// TIA Portal V17 export
// export: Created 2022-07-28T18:02:50.6515825Z, ExportSetting None, DisplayName Totally Integrated Automation Portal, DisplayVersion V17, DisplayName TIA Portal Openness, DisplayVersion V17, DisplayName TIA Portal Teamcenter Gateway, DisplayVersion V17, DisplayName TIA Portal Version Control Interface, DisplayVersion V17, DisplayName TIA Portal Test Suite Advanced, DisplayVersion V17, DisplayName SINAMICS Startdrive Advanced, DisplayVersion V17, DisplayName SINAMICS DCC, DisplayVersion V17, DisplayName SINAMICS Startdrive G130, G150, S120, S150, SINAMICS MV, S210, DisplayVersion V17, DisplayName SINAMICS Startdrive G110M, G120, G120C, G120D, G120P, G115D, DisplayVersion V17, DisplayName STEP 7 Professional, DisplayVersion V17, DisplayName SIMATIC Energy Suite, DisplayVersion V17, DisplayName STEP 7 CFC, DisplayVersion V17, DisplayName STEP 7 Safety, DisplayVersion V17, DisplayName WinCC Advanced / Unified PC, DisplayVersion V17, DisplayName SIMATIC Visualization Architect, DisplayVersion V17
FUNCTION_BLOCK "lib_fb_DSensor"   // FB18, SCL
{ S7_Optimized_Access := 'TRUE' }
AUTHOR : bean
// Descrete sensor functional block
// stored: MemoryReserve 100, SetENOAutomatically false
   VAR_INPUT
      I_Initialization { ExternalAccessible := 'False'; ExternalVisible := 'False'; ExternalWritable := 'False'} : Bool := FALSE;   // 1 = Restart PLC is active (First scan)
      I_Raw { ExternalAccessible := 'False'; ExternalVisible := 'False'; ExternalWritable := 'False'} : Bool;   // Sensor input
      II_Mode { ExternalAccessible := 'False'; ExternalVisible := 'False'; ExternalWritable := 'False'} : Int := -1;   // Check input: 0 - NO fault, 1 - NC fault, 2 - NO warning, 3 - NC warning, 4 - NO Info condition? 5 - NC Info condition
      I_GlobalRST { ExternalAccessible := 'False'; ExternalVisible := 'False'; ExternalWritable := 'False'} : Bool;   // Reset faults
      IR_CycleTime { ExternalAccessible := 'False'; ExternalVisible := 'False'; ExternalWritable := 'False'} : Real;   // PLC last cycle time
      II_Obj_ID { ExternalAccessible := 'False'; ExternalVisible := 'False'; ExternalWritable := 'False'} : Int := -1;   // Tech ID of object
   END_VAR
   VAR_OUTPUT
      Q_ProccessedVal { ExternalAccessible := 'False'; ExternalVisible := 'False'; ExternalWritable := 'False'} : Bool;   // Proccessed value by time and modes
      Q_FLT { ExternalAccessible := 'False'; ExternalVisible := 'False'; ExternalWritable := 'False'} : Bool;   // Fault is active
      Q_WRN { ExternalAccessible := 'False'; ExternalVisible := 'False'; ExternalWritable := 'False'} : Bool;   // Warning is active
      Q_INFO { ExternalAccessible := 'False'; ExternalVisible := 'False'; ExternalWritable := 'False'} : Bool;   // Info condition is active
      Q_DBReadErr { ExternalAccessible := 'False'; ExternalVisible := 'False'; ExternalWritable := 'False'} : Bool;   // Object DB reading fault
   END_VAR
   VAR_IN_OUT
      IO_PLC_CycleInfo : Variant;
   END_VAR
   VAR
      s_SimMode { ExternalAccessible := 'False'; ExternalVisible := 'False'; ExternalWritable := 'False'} : Bool;   // Simulation mode is active
      s_Suppressed { ExternalAccessible := 'False'; ExternalVisible := 'False'; ExternalWritable := 'False'} : Bool;   // Suppress fault/warning
      TON_FLT { ExternalAccessible := 'False'; ExternalVisible := 'False'; ExternalWritable := 'False'} : "Lib_FB_Timer_ON_Simple";
      EdgeError { ExternalAccessible := 'False'; ExternalVisible := 'False'; ExternalWritable := 'False'} : "Lib_FB_Edge";
      EdgeWarning { ExternalAccessible := 'False'; ExternalVisible := 'False'; ExternalWritable := 'False'} : "Lib_FB_Edge";
   END_VAR
   VAR RETAIN
      s_Obj_Retain_BUp { ExternalAccessible := 'False'; ExternalVisible := 'False'; ExternalWritable := 'False'} : Struct
         Config : "_DSensor_Config";
         s_Suppressed : Bool;   // Suppress faults
      END_STRUCT;
      s_Simulation { ExternalAccessible := 'False'; ExternalVisible := 'False'; ExternalWritable := 'False'} : Struct
         Obj_DATA_BACKUP : Struct
            Config : "_DSensor_Config";
            s_Suppressed { S7_SetPoint := 'True'} : Bool;   // Suppress faults
         END_STRUCT;
      END_STRUCT;
   END_VAR
   VAR_TEMP
      t_FltMode : Bool;   // 1 - Fault mode is active
      t_WarnMode : Bool;   // 1 - Warn mode is active
      t_InfoMode : Bool;   // 1 - Info mode is active
      t_RST_FLT : Bool;
      t_DBReadErr : Bool;   // Fault while DB reading
      ti_DBReadErr : Int;   // Fault # while DB reading
      ti_CMDLogic : Int;   // Command word for logic
      ti_NumObjDB : UInt;   // Number of DB for storage object data
      t_ObjAnyHMI : DB_ANY;   // Ref to object data
      t_ObjVarHMI : Variant;   // Ref to object data
      t_ObjAnyPLC : DB_ANY;   // Ref to object data
      t_ObjVarPLC : Variant;   // Ref to object data
      tud_DB_ShiftHMI : UInt;   // HMI object DB number shift
      tud_DB_ShiftPLC : UInt;   // PLC object DB number shift
      t_PLC_CycleInfo : "Lib_PLC_CycleInfo";
      t_Obj_HMI : "lib_udt_DSensor_HMI";
      t_Obj_PLC : "lib_udt_DSensor_PLC";
   END_VAR
BEGIN
   //Check input:
   //0 - NO fault,
   //1 - NC fault,
   //2 - NO warning,
   //3 - NC warning,
   //4 - NO Info condition,
   //5 - NC Info condition
   //
   REGION Inputs  
       //Reinit tempory variables
       REGION Reinit tempory variables


       END_REGION

       VariantGet(SRC := #IO_PLC_CycleInfo,
                  DST => #t_PLC_CycleInfo);

       //Read Object data
       //Reinit temp values
       #t_Obj_HMI := "D_ZeroTypes".DSensor_HMI;
       #t_Obj_PLC := "D_ZeroTypes".DSensor_PLC;
       #tud_DB_ShiftHMI := "D_General_ProgramDATA".ui_Shift_DBSens_HMI;
       #tud_DB_ShiftPLC := "D_General_ProgramDATA".ui_Shift_DBSens_PLC;
       #t_FltMode := false;
       #t_WarnMode := false;
       #t_InfoMode := false;

       IF #II_Obj_ID >= 0
       THEN
           #ti_NumObjDB := INT_TO_UINT(#II_Obj_ID) + #tud_DB_ShiftHMI;
           #t_ObjAnyHMI := UINT_TO_DB_ANY(#ti_NumObjDB);
           #t_ObjVarHMI := DB_ANY_TO_VARIANT(in := #t_ObjAnyHMI, err => #ti_DBReadErr);

           //If DB exist and convertion without error
           IF #ti_DBReadErr = 0
           THEN
               VariantGet(SRC := #t_ObjVarHMI,
                          DST => #t_Obj_HMI);
           ELSE
               #t_DBReadErr := true;
           END_IF;

           #ti_NumObjDB := INT_TO_UINT(#II_Obj_ID)+ #tud_DB_ShiftPLC;
           #t_ObjAnyPLC := UINT_TO_DB_ANY(#ti_NumObjDB);
           #t_ObjVarPLC := DB_ANY_TO_VARIANT(in := #t_ObjAnyPLC, err => #ti_DBReadErr);

           //If DB exist and convertion without error
           IF #ti_DBReadErr = 0
           THEN
               VariantGet(SRC := #t_ObjVarPLC,
                          DST => #t_Obj_PLC);
           ELSE
               #t_DBReadErr := true;
           END_IF;

       ELSE
           #t_DBReadErr := true;
       END_IF;


       //Read retain data if initialization is active
       IF #I_Initialization
       THEN
           #t_Obj_HMI.Config := #s_Obj_Retain_BUp.Config;
           #s_Suppressed := #s_Obj_Retain_BUp.s_Suppressed;
       END_IF;

       //Define CMD by priority
       IF #t_PLC_CycleInfo.CMD_GLOBAL <> 0
       THEN
           #ti_CMDLogic := #t_PLC_CycleInfo.CMD_GLOBAL;
       ELSE
           IF #t_Obj_HMI.CMD <> 0
           THEN
               #ti_CMDLogic := #t_Obj_HMI.CMD;
               #t_Obj_HMI.CMD := 0;
           END_IF;
       END_IF;

       #t_RST_FLT := #I_GlobalRST
       OR #t_Obj_HMI.Config.AutoReset;

       CASE #ti_CMDLogic OF
           0:  //Do nothing
               ;
           7:  //Sim mode ON
               IF NOT #s_SimMode
               THEN
                   #s_SimMode := TRUE;
                   #s_Simulation.Obj_DATA_BACKUP.Config := #t_Obj_HMI.Config;
                   #s_Simulation.Obj_DATA_BACKUP.s_Suppressed := #s_Suppressed;
               END_IF;
           8:  //Sim mode OFF
               IF #s_SimMode
               THEN
                   #s_SimMode := FALSE;
                   #t_Obj_HMI.Config := #s_Simulation.Obj_DATA_BACKUP.Config;
                   #s_Suppressed := #s_Simulation.Obj_DATA_BACKUP.s_Suppressed;
               END_IF;
           31..32://Reset faults
               #t_RST_FLT := TRUE;
           34: //Set bit for autoreset output 
               #t_Obj_HMI.Config.AutoReset := true;
           35: //Reset bit for autoreset output 
               #t_Obj_HMI.Config.AutoReset := false;
           64: //Fault/warning suppressed
               #s_Suppressed := NOT #s_Suppressed;
           80: //Discrete sensor. Invert value (Sim Mode)
               IF #s_SimMode
               THEN
                   #t_Obj_PLC.State.DisplayData := NOT #t_Obj_PLC.State.DisplayData;
               END_IF;
           ELSE//
               ;
       END_CASE;

   END_REGION

   REGION Proccess output value by mode
       #t_Obj_PLC.State.SensorValueHW := #I_Raw
       AND NOT #s_SimMode;

       CASE #II_Mode OF
           0:  //NO Fault condition
               #t_Obj_PLC.State.SensorValueLogic := #t_Obj_PLC.State.SensorValueHW;
               #t_FltMode := true;
               #t_Obj_PLC.State.SensorNO := true;
           1:  //NC Fault condition
               #t_Obj_PLC.State.SensorValueLogic := NOT #t_Obj_PLC.State.SensorValueHW;
               #t_FltMode := true;
               #t_Obj_PLC.State.SensorNO := false;
           2:  //NO Warning condition
               #t_Obj_PLC.State.SensorValueLogic := #t_Obj_PLC.State.SensorValueHW;
               #t_WarnMode := true;
               #t_Obj_PLC.State.SensorNO := true;
           3:  //NC Warning condition
               #t_Obj_PLC.State.SensorValueLogic := NOT #t_Obj_PLC.State.SensorValueHW;
               #t_WarnMode := true;
               #t_Obj_PLC.State.SensorNO := false;
           4:  //NO Info condition
               #t_Obj_PLC.State.SensorValueLogic := #t_Obj_PLC.State.SensorValueHW;
               #t_InfoMode := true;
               #t_Obj_PLC.State.SensorNO := true;
           5:  //NC Info condition
               #t_Obj_PLC.State.SensorValueLogic := NOT #t_Obj_PLC.State.SensorValueHW;
               #t_InfoMode := true;
               #t_Obj_PLC.State.SensorNO := false;
           ELSE  //
               #t_Obj_HMI := "D_ZeroTypes".DSensor_HMI;
               #t_Obj_PLC := "D_ZeroTypes".DSensor_PLC;

               IF NOT #t_DBReadErr THEN
                   VariantPut(SRC := #t_Obj_HMI,
                              DST := #t_ObjVarHMI);

                   VariantPut(SRC := #t_Obj_PLC,
                              DST := #t_ObjVarPLC);
               END_IF;

               #Q_ProccessedVal :=
               #Q_FLT :=
               #Q_WRN :=
               #Q_INFO := false;
               #Q_DBReadErr := true;

               RETURN;
       END_CASE;
       REGION Warnings and faults 
           //Time befor out detect
           #TON_FLT(IB_StartTimerInput := #t_Obj_PLC.State.SensorValueLogic,
                    IR_CycleTime := #IR_CycleTime,
                    IR_SpTime := #t_Obj_HMI.Config.WarnDetectTime);

           //Proccessed output value
           IF NOT #s_SimMode
           THEN
               #t_Obj_PLC.State.DisplayData := (#TON_FLT.QB_TimerOut
               OR (#t_Obj_PLC.State.DisplayData
               AND NOT #t_RST_FLT))
               AND NOT #s_Suppressed;
           ELSE
               #t_Obj_PLC.State.DisplayData := #t_Obj_PLC.State.DisplayData;
           END_IF;

           #t_Obj_PLC.State.SomeFlt := #t_Obj_PLC.State.DisplayData
           AND  #t_FltMode;

           #t_Obj_PLC.State.SomeWrn := #t_Obj_PLC.State.DisplayData
           AND #t_WarnMode;

           #t_Obj_PLC.State.SomeInfo := #t_Obj_PLC.State.DisplayData
           AND #t_InfoMode;

           //Excluded (suppressed) fault is active
           #t_Obj_PLC.State.SuppressedFltWrn := (#TON_FLT.QB_TimerOut
           AND #s_Suppressed);

           //New fault checking
           #EdgeError(IB_Input := #t_Obj_PLC.State.SomeFlt);
           //New warning checking
           #EdgeWarning(IB_Input := #t_Obj_PLC.State.SomeWrn);

       END_REGION
   END_REGION

   REGION PLC State + Counter
       "Lib_FC_DSens_CycleInfo_Count_State"(Alarm := #t_Obj_PLC.State.SomeFlt,
                                            AlarmNew := #EdgeError.QB_EdgePos,
                                            Warning := #t_Obj_PLC.State.SomeWrn,
                                            WarningNew := #EdgeWarning.QB_EdgePos,
                                            Simulation := #s_SimMode,
                                            PLC_CycleInfo := #t_PLC_CycleInfo);

   END_REGION

   REGION Write retain data to BUp
       //Read retain data if initialization is active
       IF NOT #I_Initialization
       THEN
           #s_Obj_Retain_BUp.Config :=  #t_Obj_HMI.Config;
           #s_Obj_Retain_BUp.s_Suppressed := #s_Suppressed;
       END_IF;
   END_REGION


   REGION Outputs
       //Outputs
       //Object DBs
       //HMI DB
       #t_Obj_HMI.CMD := 0;

       #t_Obj_HMI.ID := #II_Obj_ID;
       #t_Obj_HMI.CLSID := 40;

       //Write alarms to PLC storage
       #t_Obj_PLC.Alarm.SensorFlt := #t_Obj_PLC.State.SomeFlt;
       #t_Obj_PLC.Alarm.SensorWrn := #t_Obj_PLC.State.SomeWrn;
       #t_Obj_PLC.Alarm.SensorInfo := #t_Obj_PLC.State.SomeInfo;
       #t_Obj_PLC.Alarm.SimMode := #s_SimMode;
       #t_Obj_PLC.Alarm.NotSimMode := NOT #s_SimMode;
       #t_Obj_PLC.Alarm.Suppressed := #s_Suppressed;
       #t_Obj_PLC.Alarm.Consider := NOT #s_Suppressed;
       #t_Obj_PLC.Alarm.AutoResetEn := #t_Obj_PLC.State.AutoReset;
       #t_Obj_PLC.Alarm.AutoResetDis := NOT #t_Obj_PLC.State.AutoReset;
       #t_Obj_PLC.Alarm.SuppesedActive := #t_Obj_PLC.State.SuppressedFltWrn;

       //Write alarms to HMI
       #t_Obj_HMI.Status.w_AW1.%X0 := #t_Obj_PLC.Alarm.SensorFlt;       //х0 - Sensor Fault signal
       #t_Obj_HMI.Status.w_AW1.%X1 := #t_Obj_PLC.Alarm.SensorWrn;          //х1 - Sensor Warning signal
       #t_Obj_HMI.Status.w_AW1.%X2 := #t_Obj_PLC.Alarm.SensorInfo;         //x2 - Sensor Info signal
       #t_Obj_HMI.Status.w_AW1.%X3 := #t_Obj_PLC.Alarm.SimMode;      //x3 - Sim mode is active
       #t_Obj_HMI.Status.w_AW1.%X4 := NOT #t_Obj_PLC.Alarm.NotSimMode;  //x4 - Sim mode disabled
       #t_Obj_HMI.Status.w_AW1.%X5 := #t_Obj_PLC.Alarm.SuppesedActive; //x5 - Suppressed value is active

       #t_Obj_HMI.Status.w_AW2.%X0 := #t_Obj_PLC.Alarm.Suppressed;       //х0 - Suppress fault/warning
       #t_Obj_HMI.Status.w_AW2.%X1 := #t_Obj_PLC.Alarm.Consider;   //x1 - Consider fault/warning
       #t_Obj_HMI.Status.w_AW2.%X2 := #t_Obj_PLC.Alarm.AutoResetEn;       //х0 - Suppress fault/warning
       #t_Obj_HMI.Status.w_AW2.%X3 := #t_Obj_PLC.Alarm.AutoResetDis;   //x1 - Consider fault/warning

       //Write STW to PLC storage
       #t_Obj_PLC.State.AutoReset := #t_Obj_HMI.Config.AutoReset;
       #t_Obj_PLC.State.SimMode := #s_SimMode;
       #t_Obj_PLC.State.ReadFlt := #t_DBReadErr;
       #t_Obj_PLC.State.SuppressFltWrn := #s_Suppressed;

       //Write STW to HMI
       #t_Obj_HMI.Status.dw_STW.%X0  :=  #t_Obj_PLC.State.DisplayData;
       #t_Obj_HMI.Status.dw_STW.%X1  :=  #t_Obj_PLC.State.SimMode;
       #t_Obj_HMI.Status.dw_STW.%X2  :=  #t_Obj_PLC.State.SomeFlt;
       #t_Obj_HMI.Status.dw_STW.%X3  :=  #t_Obj_PLC.State.SomeWrn;
       #t_Obj_HMI.Status.dw_STW.%X4  :=  #t_Obj_PLC.State.SomeInfo;
       #t_Obj_HMI.Status.dw_STW.%X5  :=  #t_Obj_PLC.State.SuppressedFltWrn;
       #t_Obj_HMI.Status.dw_STW.%X6  :=  #t_Obj_PLC.State.ReadFlt;
       #t_Obj_HMI.Status.dw_STW.%X7  :=  #t_Obj_PLC.State.SuppressFltWrn;
       #t_Obj_HMI.Status.dw_STW.%X8  :=  #t_Obj_PLC.State.SensorNO;
       #t_Obj_HMI.Status.dw_STW.%X9  :=  #t_Obj_PLC.State.SensorValueLogic;
       #t_Obj_HMI.Status.dw_STW.%X10  :=  #t_Obj_PLC.State.SensorValueHW;
       #t_Obj_HMI.Status.dw_STW.%X11  :=  #t_Obj_PLC.State.AutoReset;

       //Block outputs
       #Q_ProccessedVal := #t_Obj_PLC.State.DisplayData;
       #Q_FLT := #t_Obj_PLC.State.SomeFlt;
       #Q_WRN := #t_Obj_PLC.State.SomeWrn;
       #Q_INFO := #t_Obj_PLC.State.SomeInfo;
       #Q_DBReadErr := #t_DBReadErr;

       IF NOT #t_DBReadErr THEN
           VariantPut(SRC := #t_Obj_HMI,
                      DST := #t_ObjVarHMI);

           VariantPut(SRC := #t_Obj_PLC,
                      DST := #t_ObjVarPLC);
       END_IF;

       VariantPut(SRC := #t_PLC_CycleInfo,
                  DST := #IO_PLC_CycleInfo);

   END_REGION

   //10.02.2022
END_FUNCTION_BLOCK
